(* LS Electric XG5000 project: 05_Practice4_Flicker_Upcounter *)
(* PLC LSPLC *)
(* module base 0 slot 0: 입력 모듈:XGI-D21A (DC 24V 입력, 8점 (전류소스/싱크입력)) *)
(* module base 0 slot 1: 출력 모듈:XGQ-RY1A (릴레이 출력, 8점 (2A용, 단독 COM.)) *)

PROGRAM NewProgram (* task: 스캔 프로그램 *)
VAR
    램프 AT %QX0.1.0 : BOOL;
    리셋 : BOOL;
    스위치 AT %IX0.0.0 : BOOL;
    업카운터 : CTU_INT;
    타이머1 : TON;
    타이머2 : TON;
END_VAR

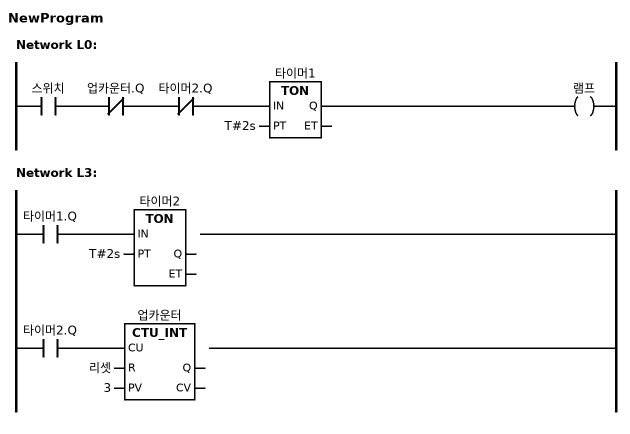
(* Rung L0 *)
타이머1(IN := 스위치 AND NOT 업카운터.Q AND NOT 타이머2.Q, PT := T#2s);
램프 := 타이머1.Q;
(* Rung L3 *)
타이머2(IN := 타이머1.Q, PT := T#2s);
업카운터(CU := 타이머2.Q, R := 리셋, PV := 3);
END_PROGRAM